RoboDK station: RobotDK_Simulation.rdk

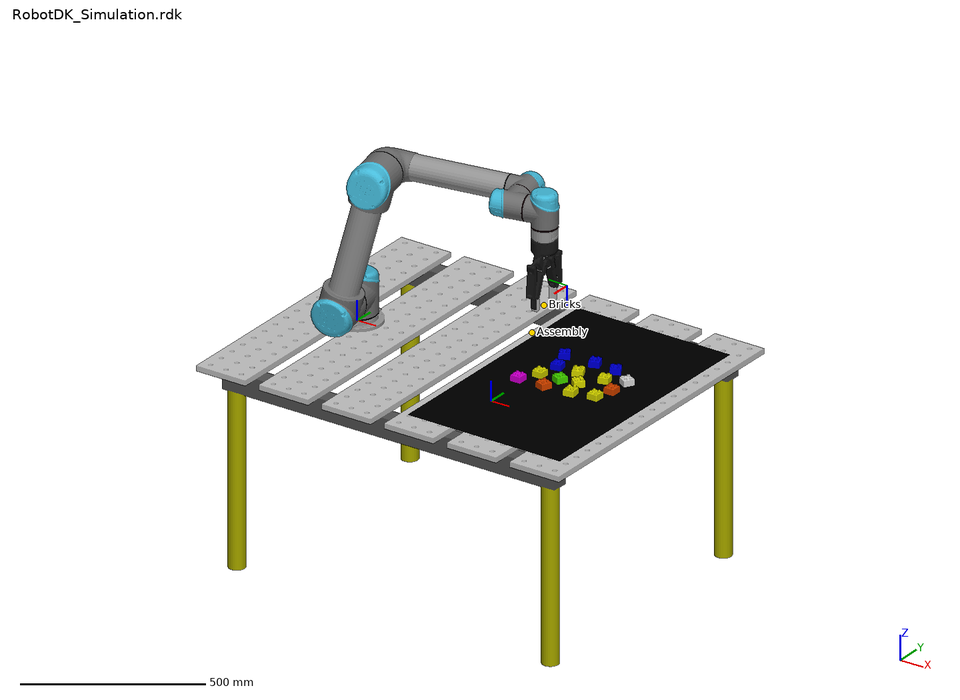
[picture v0: the station drawn from its stored meshes, robots at their saved joint values, targets as dots, program paths as lines]
Station RobotDK_Simulation (saved by RoboDK 5.5.4). Poses are relative to the parent item; angles as X-Y-Z fixed-axis rotations.
  - frame UR5 Base at (-80, 0, 0) mm
    - robot UR5: 6 axes
        modified DH rows (alpha deg, a mm, theta deg, d mm): 0, 0, 0, 89.2; 90, 0, 180, 0; 0, 425, 0, 0; 0, 392, 0, 109.3; -90, 0, 0, 94.75; 90, 0, 0, 82.5
        joint limits [-360, -360, -360, -360, -360, -360] to [360, 360, 360, 360, 360, 360]; home [0, -90, -90, 0, 90, 0]; saved at [12.252, -104.532, -77.106, -88.695, 89.786, 11.882]
      - tool Gripper, TCP at (1.74, 9.14, 189.81) mm, size 139 x 75 x 203.7 mm
      - frame Camera at (-3.41, -73.31, 121.52) mm
    - target Assembly (joint target) at (450, 180, 17.13) mm, rotated rx 180 ry 0 rz 0 deg; joints [188.768, 25.283, -116.286, 1.003, 270, 278.768] of UR5
    - target Bricks (joint target) at (601.53, 17.71, 206.36) mm, rotated rx 179.72 ry -0.28 rz -89.63 deg; joints [12.252, -104.532, -77.106, -88.695, 89.786, 11.882] of UR5
  - frame Plate at (500, -200, 0) mm
    - object LEGO_DUPLO_BRICK 8 at (220.5, 287.38, 1) mm, rotated rx 0 ry 0 rz -30.77 deg, size 31.7 x 31.7 x 23.7 mm, geometry from LEGO_DUPLO_BRICK_2X2.igs
    - object Plate at (-82.27, -163.29, 0) mm, rotated rx 90 ry 0 rz 0 deg, size 500 x 1 x 800 mm, geometry from Plate.STEP
    - object LEGO_DUPLO_BRICK 2 at (86.05, 346.09, 1) mm, rotated rx 0 ry 0 rz -68.9 deg, size 31.7 x 31.7 x 23.7 mm, geometry from LEGO_DUPLO_BRICK_2X2.igs
    - object LEGO_DUPLO_BRICK 7 at (222.84, 210.62, 1) mm, size 31.7 x 31.7 x 23.7 mm, geometry from LEGO_DUPLO_BRICK_2X2.igs
    - object LEGO_DUPLO_BRICK 9 at (171.9, 310.2, 1) mm, rotated rx 0 ry 0 rz 30.43 deg, size 31.7 x 31.7 x 23.7 mm, geometry from LEGO_DUPLO_BRICK_2X2.igs
    - object LEGO_DUPLO_BRICK 12 at (93.6, 244.38, 1) mm, rotated rx 0 ry 0 rz 24.6 deg, size 31.7 x 31.7 x 23.7 mm, geometry from LEGO_DUPLO_BRICK_2X2.igs
    - object LEGO_DUPLO_BRICK 13 at (4.68, 184.97, 1) mm, size 31.7 x 31.7 x 23.7 mm, geometry from LEGO_DUPLO_BRICK_2X2.igs
    - object LEGO_DUPLO_BRICK 6 at (173.79, 250.58, 1) mm, rotated rx 0 ry 0 rz 14.75 deg, size 31.7 x 31.7 x 23.7 mm, geometry from LEGO_DUPLO_BRICK_2X2.igs
    - object LEGO_DUPLO_BRICK 10 at (5.1, 308.72, 1) mm, rotated rx 0 ry 0 rz 30.09 deg, size 31.7 x 31.7 x 23.7 mm, geometry from LEGO_DUPLO_BRICK_2X2.igs
    - object LEGO_DUPLO_BRICK 5 at (142.37, 188.11, 1) mm, rotated rx 0 ry 0 rz 50.15 deg, size 31.7 x 31.7 x 23.7 mm, geometry from LEGO_DUPLO_BRICK_2X2.igs
    - object LEGO_DUPLO_BRICK 3 at (205.91, 156.22, 1) mm, rotated rx 0 ry 0 rz -0.96 deg, size 31.7 x 31.7 x 23.7 mm, geometry from LEGO_DUPLO_BRICK_2X2.igs
    - object LEGO_DUPLO_BRICK 4 at (140.63, 136.55, 1) mm, rotated rx 0 ry 0 rz 7.03 deg, size 31.7 x 31.7 x 23.7 mm, geometry from LEGO_DUPLO_BRICK_2X2.igs
    - object LEGO_DUPLO_BRICK 11 at (50.67, 137.17, 1) mm, rotated rx 0 ry 0 rz -20.15 deg, size 31.7 x 31.7 x 23.7 mm, geometry from LEGO_DUPLO_BRICK_2X2.igs
    - object LEGO_DUPLO_BRICK 1 at (63.3, 195.4, 1) mm, rotated rx 0 ry 0 rz -25.05 deg, size 31.7 x 31.7 x 23.7 mm, geometry from LEGO_DUPLO_BRICK_2X2.igs
    - object LEGO_DUPLO_BRICK 10 at (20.61, 247.55, 1) mm, rotated rx 0 ry 0 rz 10.69 deg, size 31.7 x 31.7 x 23.7 mm, geometry from LEGO_DUPLO_BRICK_2X2.igs
    - object LEGO_DUPLO_BRICK 7 at (-27.08, 128.85, 1) mm, size 31.7 x 31.7 x 23.7 mm, geometry from LEGO_DUPLO_BRICK_2X2.igs
  - Python program PartsToAssembly (listed below)
  - camera Camera 1
  - program Reset (1 instructions, listed below)
  - object Matrox Iris GTR Camera at (199.24, -40.48, 241.52) mm, rotated rx -180 ry 0 rz -131.84 deg, size 76.3 x 92.1 x 55 mm, geometry from Matrox-Iris-GTR-Camera.sld
  - object Table 1200x1000mm (Welding) at (320, 5.47, 0) mm, size 1193.8 x 965.2 x 609.6 mm, geometry from Table-1200x1000mm-Welding.sld

--- Python program PartsToAssembly ---
# Type help("robolink") or help("robodk") for more information
# Press F5 to run the script
# Note: you do not need to keep a copy of this file, your python script is saved with the station
from robolink import *  # API to communicate with RoboDK
from robodk import *  # basic matrix operations
from robodk.robomath import *  # import the robotics toolbox
import time
import csv
import os

# Use RoboDK API as RL
RDK = Robolink()

# Gather robot, tool and reference frames from the station
robot = RDK.Item('UR5', ITEM_TYPE_ROBOT)
tool = RDK.Item('Gripper', ITEM_TYPE_TOOL)
bricks = RDK.Item('Bricks', ITEM_TYPE_TARGET)
home = RDK.Item('Bricks', ITEM_TYPE_TARGET)
reff = RDK.Item('Assembly', ITEM_TYPE_TARGET)

# Get variable parameters
BrickW = 32
BrickH = 19
HalfBrickW = 32/2
BricksApproach = 100

# CSV position import
fig1 = []
fig2 = []
fig3 = []
fig4 = []
fig5 = []

# Reading the .csv files
def read_csv(filename, fig):
    with open(filename, 'r') as csvfile:
        csvreader = csv.reader(csvfile)
        next(csvreader)  # Skip the first row, because of the x,y,angle
        for row in csvreader:
            fig.append([float(val) for val in row[1:]])

# Calling for the fig .csv
read_csv('fig1.csv', fig1)
read_csv('fig2.csv', fig2)
read_csv('fig3.csv', fig3)
read_csv('fig4.csv', fig4)
read_csv('fig5.csv', fig5)

# Creating one big matrix with all of the data
Figs = [fig1, fig2, fig3, fig4, fig5]

# End location of the robot - This is where the robot is assembling the figures.
# It makes a half a brick space between each figure.
EndLocation = []
for i in range(len(Figs)):
    EndLocation.append(reff.Pose()*transl(0,(BrickW+HalfBrickW)*i,0))

# Tool setup - ON/OFF - For the simulation, it is different in the real word application
def TCP_On(toolitem):
    """Attaches the closest object to the toolitem Htool pose,
    It will also output appropriate function calls on the generated robot program (call to TCP_On)"""
    robot.setDO(0, 0)
    pause(0.005)
    toolitem.AttachClosest()
    # toolitem.RDK().RunMessage('Set air valve on')
    toolitem.RDK().RunProgram('TCP_On()');
    robot.setDO(0, 1)


def TCP_Off(toolitem, itemleave=0):
    """Detaches the closest object attached to the toolitem Htool pose,
    It will also output appropriate function calls on the generated robot program (call to TCP_Off)"""
    # toolitem.DetachClosest(itemleave)
    robot.setDO(0, 1)
    pause(0.005)
    toolitem.DetachAll(itemleave)
    # toolitem.RDK().RunMessage('Set air valve off')
    toolitem.RDK().RunProgram('TCP_Off()');
    robot.setDO(0, 0)

# Use this to make the code run faster
RDK.Render(False)

# Define position of bricks - Taking the position of each brick from the Figs matrix, and transfering degrees to rads
FigLocs = []
for x in range(len(Figs)):
    Loc = []
    for i in range(len(Figs[x])):
        location = reff.Pose()*transl(Figs[x][i][0],Figs[x][i][1],Figs[x][i][2])*rotz((Figs[x][i][3] * pi)/180)
        # If the line above is not working, try these
        #location = reff.Pose() * transl(float(Figs[x][i][0]), float(Figs[x][i][1]), float(Figs[x][i][2])) * rotz(float(Figs[x][i][3]*3.14159265359)/180)
        #location = reff.Pose() * transl(Figs[x][i][0][0], Figs[x][i][1][0], Figs[x][i][2][0]) * rotz(Figs[x][i][3][0]*3.14159265359)/180
        Loc.append(location)
    FigLocs.append(Loc)

# Running through this cycle, until it assembles all of the figures.
for x in range(len(FigLocs)):
    for i in range(len(FigLocs[x])):
        #Pick up
        approach = FigLocs[x][i]*transl(0,0,-BricksApproach)
        robot.MoveL(approach)
        robot.MoveL(FigLocs[x][i])
        TCP_On(tool)
        # Use this with the real robot
        #robot.setDO(4, 1)
        #time.sleep(0.1)
        #robot.setDO(4, 0)
        robot.MoveJ(approach)

        #Place
        Approach = EndLocation[x]*transl(0,0,-BricksApproach+(-BrickH*i))
        robot.MoveL(Approach)
        robot.MoveL(EndLocation[x]*transl(0,0,-BrickH*i))
        TCP_Off(tool)
        # Use this with the real robot
        #robot.setDO(5, 1)
        #time.sleep(0.1)
        #robot.setDO(5, 0)
        robot.MoveJ(Approach)

# Reset position of robot
robot.MoveJ(home)

--- program Reset (robot UR5) ---
  Replace objects
